// SIMATIC S7-200 SMART project (STEP 7-Micro/WIN SMART), CPU SR40

ORGANIZATION_BLOCK MAIN:OB1
TITLE=程序注释
BEGIN
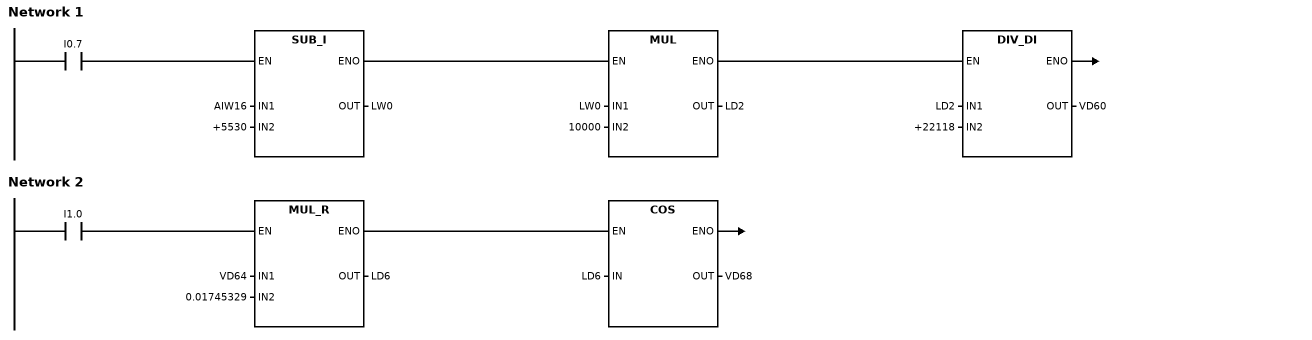
Network 1
LD     I0.7
MOVW   AIW16, LW0
AENO
-I     +5530, LW0
AENO
MOVW   LW0, LW4
AENO
MUL    10000, LD2
AENO
MOVD   LD2, VD60
/D     +22118, VD60
Network 2
LD     I1.0
MOVR   VD64, LD6
AENO
*R     0.01745329, LD6
AENO
COS    LD6, VD68
END_ORGANIZATION_BLOCK
